Fanuc KAREL source: IO0225.KL

-- PROVISIONAL review KL for V770-1; original PC SHA256 30372dfdce83099aee3e9a24a129908d8fe4fc2e2b8fe93463dd8997e33dd093
-- Incomplete behavior may be omitted. Consult companion uncertainty JSON. Do not deploy.
PROGRAM IO0225
%NOLOCKGROUP
-- UNRESOLVED_LOCAL_POOL 5 cells at code offset 13; source declarations unknown
-- DIRECT_LOCAL_WORD_ACCESS alone does not prove INTEGER, REAL, or BOOLEAN
BEGIN
  -- UNRESOLVED_PC offsets 0-18; opcodes 2B,2C,7B
  -- UNRESOLVED_PC offsets 23-30; opcodes 9D,23
  -- UNRESOLVED_PC offsets 35-49; opcodes 2E,22,9D,33,35
  -- UNRESOLVED_PC offsets 54-61; opcodes 9D,23
  -- UNRESOLVED_PC offsets 66-77; opcodes 2E,23
  -- UNRESOLVED_PC offsets 82-129; opcodes 27,22,27,3F,27,3F,22,22,AF
  -- UNRESOLVED_PC offsets 134-138; opcodes 7F
  -- UNRESOLVED_PC offsets 143-147; opcodes 27,AA
  -- UNRESOLVED_PC offsets 152-156; opcodes 7F
END IO0225
